{attribute addProperty BoxType "ELX4181-0000-0016"}
{attribute addProperty Id "Ch_1Ch_1_10CBEF651620WcStateAT %I*WcState_28A8677510.1250InfoDataAT %I*InfoData_275E3363128160"}
{attribute addProperty CRC "62645213"}
{attribute addProperty SizeInBites "145"}
{attribute addProperty SizeInBytes "18.125"}
TYPE ELX4181_F21B7298 :
STRUCT
	{attribute addProperty Name "Ch_1"}
	Ch_1 : Ch_1_10CBEF65;
	{attribute addProperty Name "WcState"}
	WcState : WcState_28A86775;
	{attribute addProperty Name "InfoData"}
	InfoData : InfoData_275E3363;
END_STRUCT
END_TYPE

(* stored: Version 1.2.0.0, ProductVersion 3.1.4024.9
   DUT ELX4181_F21B7298: Id {2448b8ee-fc44-4a2d-83db-74116853fc94} *)
